(* PLC project Unnamed, Unknown Unnamed 1 *)
(* stored: creationDateTime 2026-05-04T00:14:33, modificationDateTime 2026-05-04T00:14:33 *)

(* simple boolean *)
PROGRAM main
  VAR
    InputA : BOOL := TRUE;
    InputB : BOOL := FALSE;
    Result : BOOL := FALSE;
  END_VAR

            Result := InputA AND NOT InputB;
          
END_PROGRAM

CONFIGURATION Config0
  RESOURCE Res0 ON PLC
    TASK task0(INTERVAL := T#20ms, PRIORITY := 1);
    PROGRAM instance0 WITH task0 : main;
  END_RESOURCE
END_CONFIGURATION
